// TIA Portal V20 export
TYPE "LKinCtrl_PointEditor_typePointTableExternalEvents"
// stored: Access Published
   STRUCT
      selectionChanged { ExternalAccessible := 'False'; ExternalVisible := 'False'; ExternalWritable := 'False'} : Struct
         trigger : Bool;   // triggers event. Only true for 1 cycle.
         noSelection : Bool;
         selectedIndex : DInt;
      END_STRUCT;
   END_STRUCT;
END_TYPE
